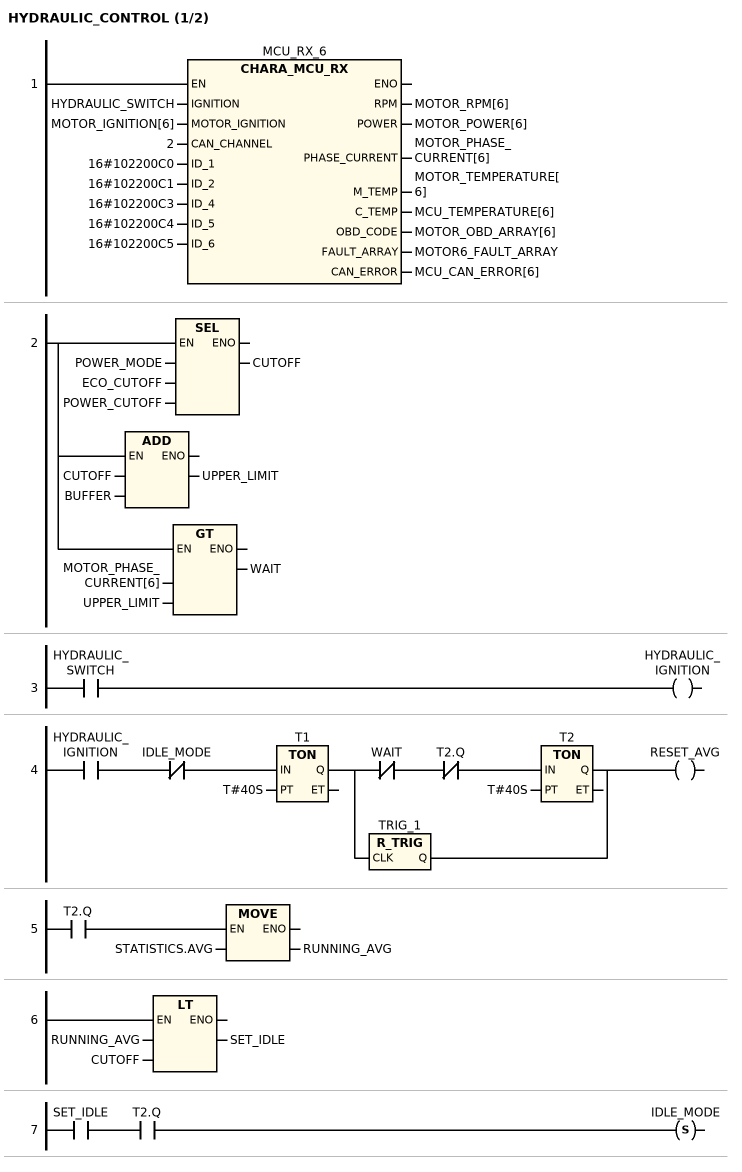
[picture p24: HYDRAULIC_CONTROL (LD)]
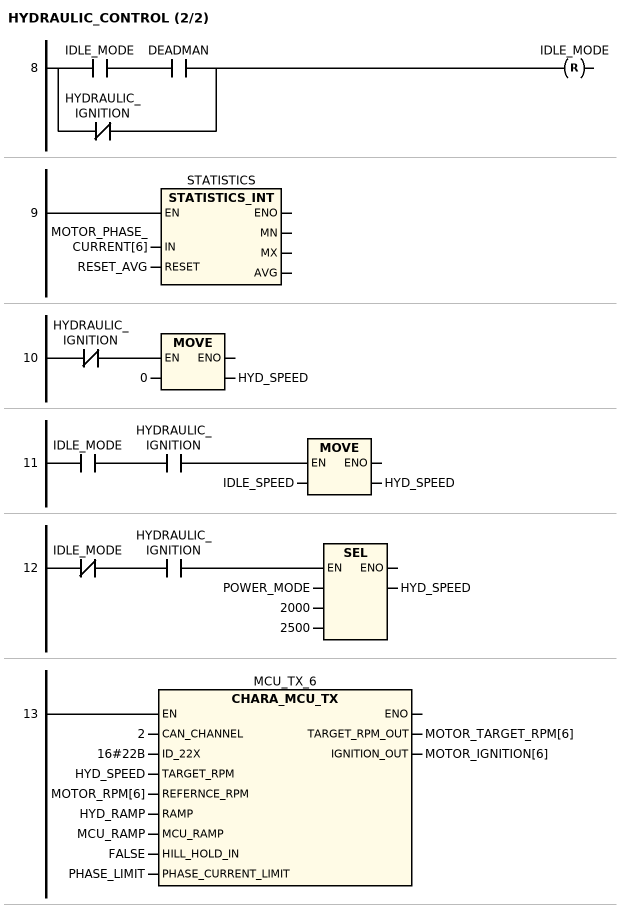
_LD_ (* Ladder Diagram *)
NETWORK 1
	*
		EN --- MCU_RX_6:CHARA_MCU_RX(IGNITION: HYDRAULIC_SWITCH, MOTOR_IGNITION: MOTOR_IGNITION[6], CAN_CHANNEL: 2, ID_1: 16#102200C0, ID_2: 16#102200C1, ID_4: 16#102200C3, ID_5: 16#102200C4, ID_6: 16#102200C5, POWER => MOTOR_POWER[6], PHASE_CURRENT => MOTOR_PHASE_CURRENT[6], M_TEMP => MOTOR_TEMPERATURE[6], C_TEMP => MCU_TEMPERATURE[6], OBD_CODE => MOTOR_OBD_ARRAY[6], FAULT_ARRAY => MOTOR6_FAULT_ARRAY, CAN_ERROR => MCU_CAN_ERROR[6]) => MOTOR_RPM[6]
NETWORK 2
	*
		EN --- SEL(POWER_MODE, ECO_CUTOFF, POWER_CUTOFF) => CUTOFF
		EN --- ADD(CUTOFF, BUFFER) => UPPER_LIMIT
		EN --- GT(MOTOR_PHASE_CURRENT[6], UPPER_LIMIT) => WAIT
NETWORK 3
	[HYDRAULIC_SWITCH] --- (HYDRAULIC_IGNITION)
NETWORK 4
	[HYDRAULIC_IGNITION] - [/IDLE_MODE] - T1:TON(IN: *, PT: T#40S) - { [/WAIT] - [/T2.Q] - T2:TON(IN: *, PT: T#40S) | TRIG_1:R_TRIG(CLK: *) } --- (RESET_AVG)
NETWORK 5
	[T2.Q]
		EN --- MOVE(STATISTICS.AVG) => RUNNING_AVG
NETWORK 6
	*
		EN --- LT(RUNNING_AVG, CUTOFF) => SET_IDLE
NETWORK 7
	[SET_IDLE] - [T2.Q] --- (S IDLE_MODE)
NETWORK 8
	{ [IDLE_MODE] - [DEADMAN] | [/HYDRAULIC_IGNITION] } --- (R IDLE_MODE)
NETWORK 9
	*
		EN --- STATISTICS:STATISTICS_INT(IN: MOTOR_PHASE_CURRENT[6], RESET: RESET_AVG)
NETWORK 10
	[/HYDRAULIC_IGNITION]
		EN --- MOVE(0) => HYD_SPEED
NETWORK 11
	[IDLE_MODE] - [HYDRAULIC_IGNITION]
		EN --- MOVE(IDLE_SPEED) => HYD_SPEED
NETWORK 12
	[/IDLE_MODE] - [HYDRAULIC_IGNITION]
		EN --- SEL(POWER_MODE, 2000, 2500) => HYD_SPEED
NETWORK 13
	*
		EN --- MCU_TX_6:CHARA_MCU_TX(CAN_CHANNEL: 2, ID_22X: 16#22B, TARGET_RPM: HYD_SPEED, REFERNCE_RPM: MOTOR_RPM[6], RAMP: HYD_RAMP, MCU_RAMP: MCU_RAMP, HILL_HOLD_IN: FALSE, PHASE_CURRENT_LIMIT: PHASE_LIMIT, IGNITION_OUT => MOTOR_IGNITION[6]) => MOTOR_TARGET_RPM[6]
_END_LD_
(* the same logic as Structured Text *)
(* Network 1 *)
MCU_RX_6(IGNITION := HYDRAULIC_SWITCH, MOTOR_IGNITION := MOTOR_IGNITION[6], CAN_CHANNEL := 2, ID_1 := 16#102200C0, ID_2 := 16#102200C1, ID_4 := 16#102200C3, ID_5 := 16#102200C4, ID_6 := 16#102200C5);
MOTOR_POWER[6] := MCU_RX_6.POWER;
MOTOR_PHASE_CURRENT[6] := MCU_RX_6.PHASE_CURRENT;
MOTOR_TEMPERATURE[6] := MCU_RX_6.M_TEMP;
MCU_TEMPERATURE[6] := MCU_RX_6.C_TEMP;
MOTOR_OBD_ARRAY[6] := MCU_RX_6.OBD_CODE;
MOTOR6_FAULT_ARRAY := MCU_RX_6.FAULT_ARRAY;
MCU_CAN_ERROR[6] := MCU_RX_6.CAN_ERROR;
MOTOR_RPM[6] := MCU_RX_6.RPM;
(* Network 2 *)
CUTOFF := SEL(POWER_MODE, ECO_CUTOFF, POWER_CUTOFF);
UPPER_LIMIT := CUTOFF + BUFFER;
WAIT := MOTOR_PHASE_CURRENT[6] > UPPER_LIMIT;
(* Network 3 *)
HYDRAULIC_IGNITION := HYDRAULIC_SWITCH;
(* Network 4 *)
T1(IN := HYDRAULIC_IGNITION AND NOT IDLE_MODE, PT := T#40S);
T2(IN := T1.Q AND NOT WAIT AND NOT T2.Q, PT := T#40S);
TRIG_1(CLK := T1.Q);
RESET_AVG := T2.Q OR TRIG_1.Q;
(* Network 5 *)
IF T2.Q THEN
	RUNNING_AVG := STATISTICS.AVG;
END_IF;
(* Network 6 *)
SET_IDLE := RUNNING_AVG < CUTOFF;
(* Network 7 *)
IF SET_IDLE AND T2.Q THEN IDLE_MODE := TRUE; END_IF;
(* Network 8 *)
IF IDLE_MODE AND DEADMAN OR NOT HYDRAULIC_IGNITION THEN IDLE_MODE := FALSE; END_IF;
(* Network 9 *)
STATISTICS(IN := MOTOR_PHASE_CURRENT[6], RESET := RESET_AVG);
(* Network 10 *)
IF NOT HYDRAULIC_IGNITION THEN
	HYD_SPEED := 0;
END_IF;
(* Network 11 *)
IF IDLE_MODE AND HYDRAULIC_IGNITION THEN
	HYD_SPEED := IDLE_SPEED;
END_IF;
(* Network 12 *)
IF NOT IDLE_MODE AND HYDRAULIC_IGNITION THEN
	HYD_SPEED := SEL(POWER_MODE, 2000, 2500);
END_IF;
(* Network 13 *)
MCU_TX_6(CAN_CHANNEL := 2, ID_22X := 16#22B, TARGET_RPM := HYD_SPEED, REFERNCE_RPM := MOTOR_RPM[6], RAMP := HYD_RAMP, MCU_RAMP := MCU_RAMP, HILL_HOLD_IN := FALSE, PHASE_CURRENT_LIMIT := PHASE_LIMIT);
MOTOR_IGNITION[6] := MCU_TX_6.IGNITION_OUT;
MOTOR_TARGET_RPM[6] := MCU_TX_6.TARGET_RPM_OUT;
END_FUNCTION_BLOCK

(* POU MCU/CHARA_MCU_RX, LD *)
FUNCTION_BLOCK CHARA_MCU_RX
(*
Created by: Bhagyesh Unadkat
Date: 11-09-24
Version: 5
Updated by: Karthik
Update date: 08-03-25
Description: This block receives CAN data from CHARA MCU.

		***Updates***
V2
	DC current and POWER added.
V3   
	Added OBD Code and adjusted the fault array accordingly.
	CAN error added to OBD code MSB bit as it is 12-bit value.
V4 
	Taken Motor Ignition as VAR_INPUT to reset RPM AND POWER TO 0
V5
	Converted CURRENT raw values from word to int, and then dividing by 1000.
V6
	Unmerged CAN error and OBD code.
V7
	Making OBD code zero when theres is a CAN error. 

FAULT ARRAY [DATATYPE: BYTE]
[1] MSG-2 BYTE2 and MSG-5 BYTE3		
		BYTE [BIT 0..7]: MSG2BYTE2 (BIT_0 TO BIT_2)------- AND-------- MSG5BYTE3 (BIT_0 TO BIT_4)
[2] MSG 2 :BYTE 7
[3] MSG 5: BYTE 2
[4] MSG 5: BYTE 4
*)
VAR_INPUT
	IGNITION: BOOL;
	MOTOR_IGNITION: BOOL;
	CAN_CHANNEL: BYTE;
	ID_1: DWORD;
	ID_2: DWORD;
	ID_4: DWORD;
	ID_5: DWORD;
	ID_6: DWORD;
END_VAR
VAR_OUTPUT
	RPM: INT;
	POWER: INT;
	PHASE_CURRENT: WORD;
	M_TEMP: BYTE;
	C_TEMP: BYTE;
	OBD_CODE: WORD;
	FAULT_ARRAY: ARRAY [1..4] OF BYTE;
	CAN_ERROR: BOOL;
END_VAR
VAR
	RX_1: RX_CAN;
	RX_2: RX_CAN;
	RX_4: RX_CAN;
	RX_5: RX_CAN;
	RX_6: RX_CAN;
	TIMER_ERROR: TON;

	RPM_WORD: WORD;
	PHASE_WORD: WORD;
	REVERSE_DIRECTION: BOOL;
	DIR_FACTOR: INT;
	DELAY: TON;
	RPM_INT: INT;
	CURRENT_WORD: WORD;
	CURRENT_INT: INT;
	VOLTAGE_INT: INT;
	RPM_SIGNED: INT;
	POWER_INT: INT;
END_VAR
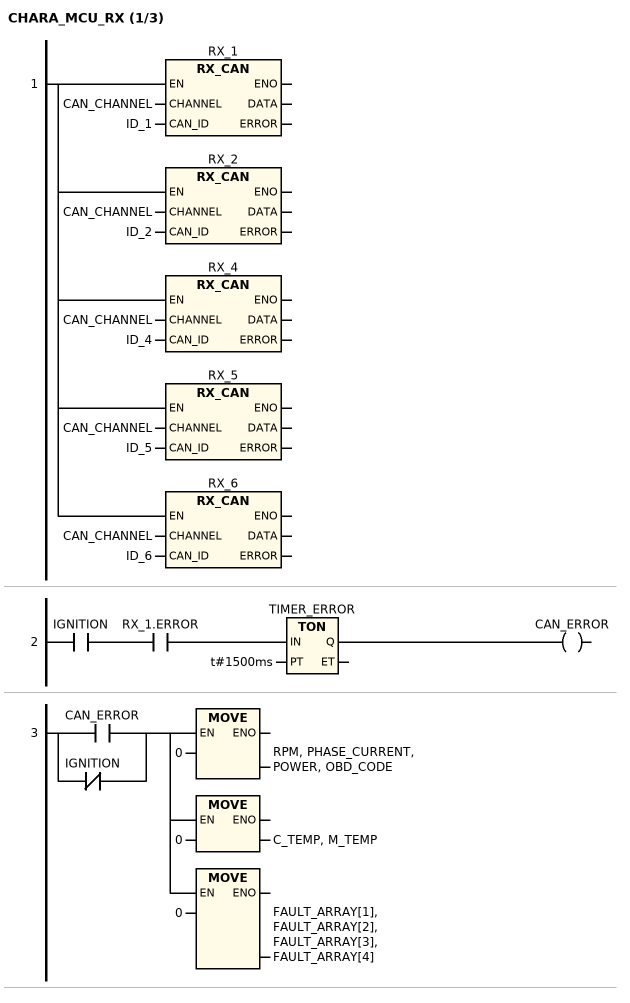
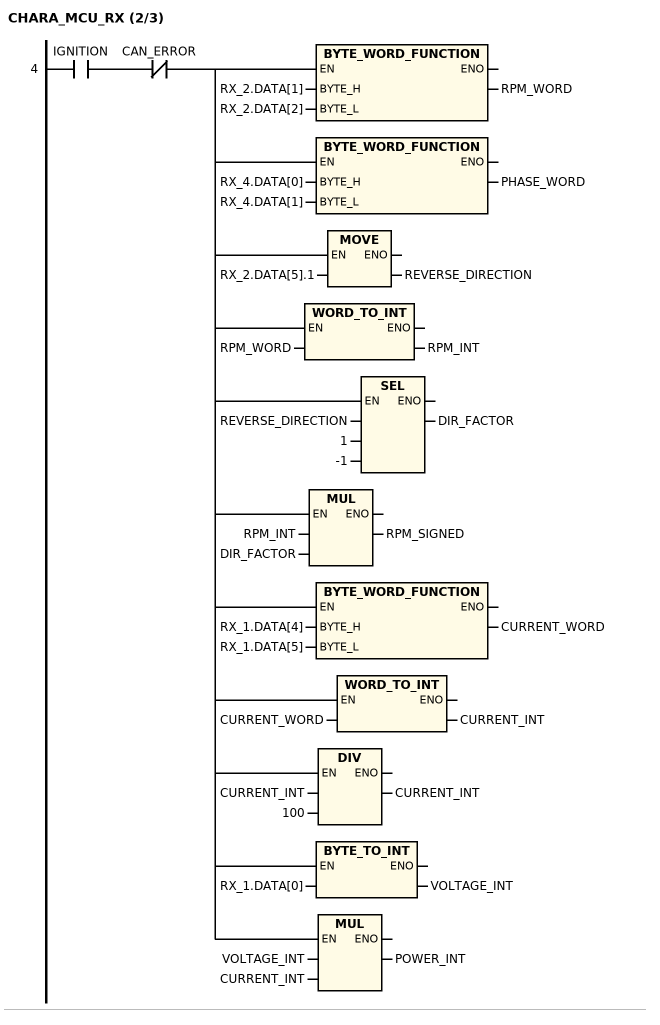
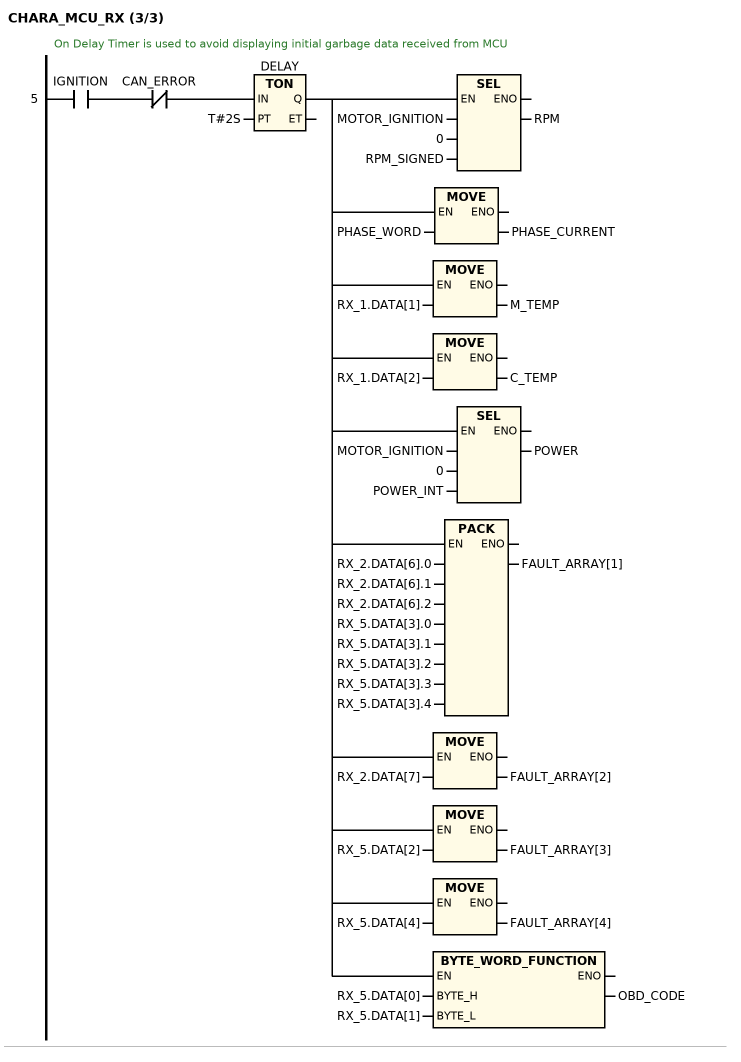
_LD_ (* Ladder Diagram *)
NETWORK 1
	*
		EN --- RX_1:RX_CAN(CHANNEL: CAN_CHANNEL, CAN_ID: ID_1)
		EN --- RX_2:RX_CAN(CHANNEL: CAN_CHANNEL, CAN_ID: ID_2)
		EN --- RX_4:RX_CAN(CHANNEL: CAN_CHANNEL, CAN_ID: ID_4)
		EN --- RX_5:RX_CAN(CHANNEL: CAN_CHANNEL, CAN_ID: ID_5)
		EN --- RX_6:RX_CAN(CHANNEL: CAN_CHANNEL, CAN_ID: ID_6)
NETWORK 2
	[IGNITION] - [RX_1.ERROR] - TIMER_ERROR:TON(IN: *, PT: t#1500ms) --- (CAN_ERROR)
NETWORK 3
	{ [CAN_ERROR] | [/IGNITION] }
		EN --- MOVE(0) => RPM, PHASE_CURRENT, POWER, OBD_CODE
		EN --- MOVE(0) => C_TEMP, M_TEMP
		EN --- MOVE(0) => FAULT_ARRAY[1], FAULT_ARRAY[2], FAULT_ARRAY[3], FAULT_ARRAY[4]
NETWORK 4
	[IGNITION] - [/CAN_ERROR]
		EN --- BYTE_WORD_FUNCTION(BYTE_H: RX_2.DATA[1], BYTE_L: RX_2.DATA[2]) => RPM_WORD
		EN --- BYTE_WORD_FUNCTION(BYTE_H: RX_4.DATA[0], BYTE_L: RX_4.DATA[1]) => PHASE_WORD
		EN --- MOVE(RX_2.DATA[5].1) => REVERSE_DIRECTION
		EN --- WORD_TO_INT(RPM_WORD) => RPM_INT
		EN --- SEL(REVERSE_DIRECTION, 1, -1) => DIR_FACTOR
		EN --- MUL(RPM_INT, DIR_FACTOR) => RPM_SIGNED
		EN --- BYTE_WORD_FUNCTION(BYTE_H: RX_1.DATA[4], BYTE_L: RX_1.DATA[5]) => CURRENT_WORD
		EN --- WORD_TO_INT(CURRENT_WORD) => CURRENT_INT
		EN --- DIV(CURRENT_INT, 100) => CURRENT_INT
		EN --- BYTE_TO_INT(RX_1.DATA[0]) => VOLTAGE_INT
		EN --- MUL(VOLTAGE_INT, CURRENT_INT) => POWER_INT
NETWORK 5 (* On Delay Timer is used to avoid displaying initial garbage data received from MCU *)
	[IGNITION] - [/CAN_ERROR] - DELAY:TON(IN: *, PT: T#2S)
		EN --- SEL(MOTOR_IGNITION, 0, RPM_SIGNED) => RPM
		EN --- MOVE(PHASE_WORD) => PHASE_CURRENT
		EN --- MOVE(RX_1.DATA[1]) => M_TEMP
		EN --- MOVE(RX_1.DATA[2]) => C_TEMP
		EN --- SEL(MOTOR_IGNITION, 0, POWER_INT) => POWER
		EN --- PACK(RX_2.DATA[6].0, RX_2.DATA[6].1, RX_2.DATA[6].2, RX_5.DATA[3].0, RX_5.DATA[3].1, RX_5.DATA[3].2, RX_5.DATA[3].3, RX_5.DATA[3].4) => FAULT_ARRAY[1]
		EN --- MOVE(RX_2.DATA[7]) => FAULT_ARRAY[2]
		EN --- MOVE(RX_5.DATA[2]) => FAULT_ARRAY[3]
		EN --- MOVE(RX_5.DATA[4]) => FAULT_ARRAY[4]
		EN --- BYTE_WORD_FUNCTION(BYTE_H: RX_5.DATA[0], BYTE_L: RX_5.DATA[1]) => OBD_CODE
_END_LD_
(* the same logic as Structured Text *)
(* Network 1 *)
RX_1(CHANNEL := CAN_CHANNEL, CAN_ID := ID_1);
RX_2(CHANNEL := CAN_CHANNEL, CAN_ID := ID_2);
RX_4(CHANNEL := CAN_CHANNEL, CAN_ID := ID_4);
RX_5(CHANNEL := CAN_CHANNEL, CAN_ID := ID_5);
RX_6(CHANNEL := CAN_CHANNEL, CAN_ID := ID_6);
(* Network 2 *)
TIMER_ERROR(IN := IGNITION AND RX_1.ERROR, PT := t#1500ms);
CAN_ERROR := TIMER_ERROR.Q;
(* Network 3: see the listing above *)
(* Network 4 *)
IF IGNITION AND NOT CAN_ERROR THEN
	RPM_WORD := BYTE_WORD_FUNCTION(BYTE_H := RX_2.DATA[1], BYTE_L := RX_2.DATA[2]);
	PHASE_WORD := BYTE_WORD_FUNCTION(BYTE_H := RX_4.DATA[0], BYTE_L := RX_4.DATA[1]);
	REVERSE_DIRECTION := RX_2.DATA[5].1;
	RPM_INT := WORD_TO_INT(RPM_WORD);
	DIR_FACTOR := SEL(REVERSE_DIRECTION, 1, -1);
	RPM_SIGNED := RPM_INT * DIR_FACTOR;
	CURRENT_WORD := BYTE_WORD_FUNCTION(BYTE_H := RX_1.DATA[4], BYTE_L := RX_1.DATA[5]);
	CURRENT_INT := WORD_TO_INT(CURRENT_WORD);
	CURRENT_INT := CURRENT_INT / 100;
	VOLTAGE_INT := BYTE_TO_INT(RX_1.DATA[0]);
	POWER_INT := VOLTAGE_INT * CURRENT_INT;
END_IF;
(* Network 5 *)
DELAY(IN := IGNITION AND NOT CAN_ERROR, PT := T#2S);
IF DELAY.Q THEN
	RPM := SEL(MOTOR_IGNITION, 0, RPM_SIGNED);
	PHASE_CURRENT := PHASE_WORD;
	M_TEMP := RX_1.DATA[1];
	C_TEMP := RX_1.DATA[2];
	POWER := SEL(MOTOR_IGNITION, 0, POWER_INT);
	FAULT_ARRAY[1] := PACK(RX_2.DATA[6].0, RX_2.DATA[6].1, RX_2.DATA[6].2, RX_5.DATA[3].0, RX_5.DATA[3].1, RX_5.DATA[3].2, RX_5.DATA[3].3, RX_5.DATA[3].4);
	FAULT_ARRAY[2] := RX_2.DATA[7];
	FAULT_ARRAY[3] := RX_5.DATA[2];
	FAULT_ARRAY[4] := RX_5.DATA[4];
	OBD_CODE := BYTE_WORD_FUNCTION(BYTE_H := RX_5.DATA[0], BYTE_L := RX_5.DATA[1]);
END_IF;
END_FUNCTION_BLOCK

(* POU MCU/CHARA_MCU_TX, LD *)
FUNCTION_BLOCK CHARA_MCU_TX
(*
Created by: Bhagyesh Unadkat
Date: Sep 11, 2024
Version: 4
Updated by: Bhagyesh
Update date: Dec 13, 2024
Description: This block transmits CAN data to the CHARA MCU to control the motor.

NOTE:  BIG ENDIAN FORMAT

Byte0 & Byte1: Signed RPM Big Endian format (-6000 to 6000)
Byte2: Ignition State =  0 & 1 (OFF and ON respectively)
Byte3: Phase Current Limit (%) = 0 - 100
Byte4: Regen (%) = 0 - 100 (Not configured yet)
Byte5: Acceleration time (s) = 1 unit is 100ms
Byte6: Deceleration time (s) =  1 unit is 100ms

CAN ID X value for the different Node ID:
41 - 9		42 - A 		43-B
	
	***UPDATES***
V2:
1. RPM transmit delay has been added after Ignition turns on..
2. CAN_TX block has been changerd to CAN_TX_ENH.
3. Temporary Phase current limit has been added to var input
V3
1. Added Ignition state bit as VAR_OUTPUT.
V4
1. UPDATED AVG RPM TO 75 TO HOLD ON THE MCU.
2. RPM DELAY TIME REDUCED TO 250MS
*)
VAR_INPUT
	CAN_CHANNEL: BYTE;
	ID_22X: DWORD;
	TARGET_RPM: INT;
	REFERNCE_RPM: INT;
	RAMP: INT;
	MCU_RAMP: BYTE;
	HILL_HOLD_IN: BOOL;
	PHASE_CURRENT_LIMIT: BYTE;
END_VAR
VAR
	IGNITION_ON: BOOL;
	IGNITION_STATE: BYTE;
	HOLD_ON: BOOL;
	ABS_RPM: INT;
	RPM_RAMP: RAMP_INT;
	WB_TARGET_RPM: WORD_BYTE_CONVERSION;
	PACK_TX: PACK_BYTES;
	TX: CAN_TX_ENH;
	RPM_DELAY: TON;
	TIMER: TON;
END_VAR
VAR_OUTPUT
	TARGET_RPM_OUT: INT;
	IGNITION_OUT: BOOL;
END_VAR
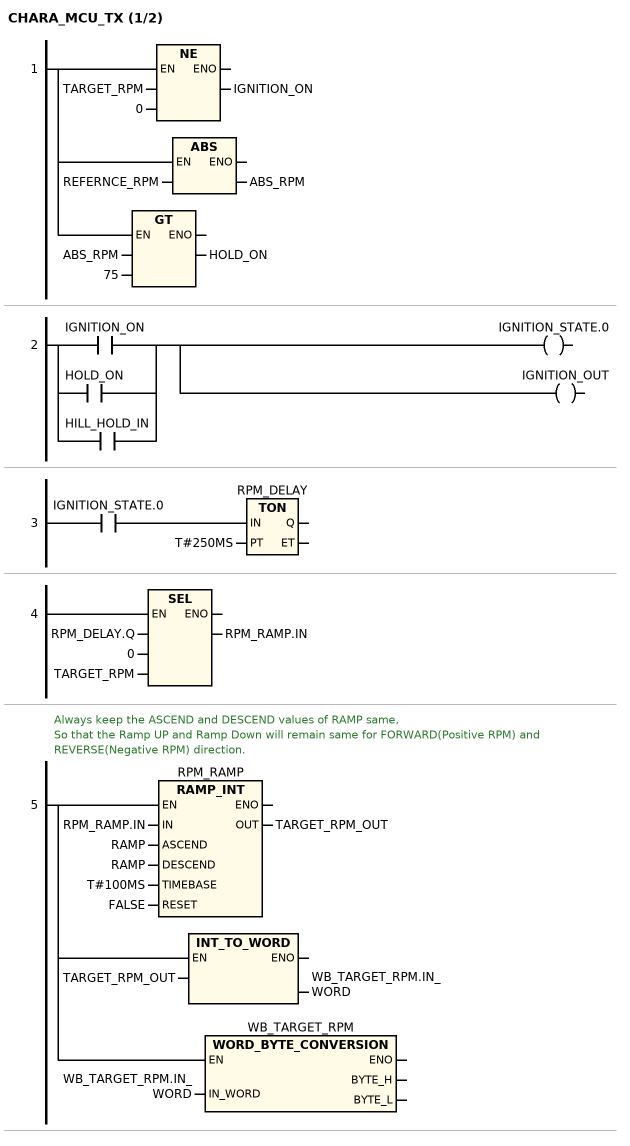
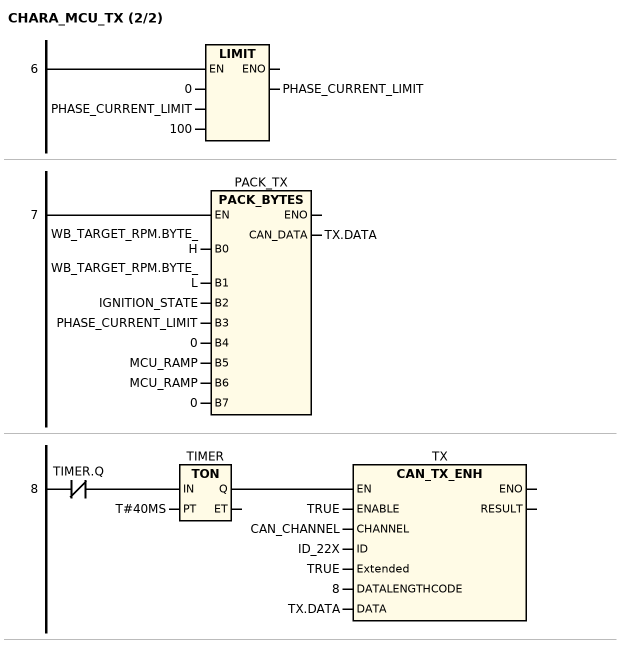
_LD_ (* Ladder Diagram *)
NETWORK 1
	*
		EN --- NE(TARGET_RPM, 0) => IGNITION_ON
		EN --- ABS(REFERNCE_RPM) => ABS_RPM
		EN --- GT(ABS_RPM, 75) => HOLD_ON
NETWORK 2
	{ [IGNITION_ON] | [HOLD_ON] | [HILL_HOLD_IN] } --- (IGNITION_STATE.0) (IGNITION_OUT)
NETWORK 3
	[IGNITION_STATE.0] - RPM_DELAY:TON(IN: *, PT: T#250MS)
NETWORK 4
	*
		EN --- SEL(RPM_DELAY.Q, 0, TARGET_RPM) => RPM_RAMP.IN
NETWORK 5 (* Always keep the ASCEND and DESCEND values of RAMP same, / So that the Ramp UP and Ramp Down will remain same for FORWARD(Positive RPM) and REVERSE(Negative RPM) direction. *)
	*
		EN --- RPM_RAMP:RAMP_INT(IN: RPM_RAMP.IN, ASCEND: RAMP, DESCEND: RAMP, TIMEBASE: T#100MS, RESET: FALSE) => TARGET_RPM_OUT
		EN --- INT_TO_WORD(TARGET_RPM_OUT) => WB_TARGET_RPM.IN_WORD
		EN --- WB_TARGET_RPM:WORD_BYTE_CONVERSION(IN_WORD: WB_TARGET_RPM.IN_WORD)
NETWORK 6
	*
		EN --- LIMIT(0, PHASE_CURRENT_LIMIT, 100) => PHASE_CURRENT_LIMIT
NETWORK 7
	*
		EN --- PACK_TX:PACK_BYTES(B0: WB_TARGET_RPM.BYTE_H, B1: WB_TARGET_RPM.BYTE_L, B2: IGNITION_STATE, B3: PHASE_CURRENT_LIMIT, B4: 0, B5: MCU_RAMP, B6: MCU_RAMP, B7: 0) => TX.DATA
NETWORK 8
	[/TIMER.Q] - TIMER:TON(IN: *, PT: T#40MS)
		EN --- TX:CAN_TX_ENH(ENABLE: TRUE, CHANNEL: CAN_CHANNEL, ID: ID_22X, Extended: TRUE, DATALENGTHCODE: 8, DATA: TX.DATA)
_END_LD_
(* the same logic as Structured Text *)
(* Network 1 *)
IGNITION_ON := TARGET_RPM <> 0;
ABS_RPM := ABS(REFERNCE_RPM);
HOLD_ON := ABS_RPM > 75;
(* Network 2 *)
IGNITION_STATE.0 := IGNITION_ON OR HOLD_ON OR HILL_HOLD_IN;
IGNITION_OUT := IGNITION_STATE.0;
(* Network 3 *)
RPM_DELAY(IN := IGNITION_STATE.0, PT := T#250MS);
(* Network 4 *)
RPM_RAMP.IN := SEL(RPM_DELAY.Q, 0, TARGET_RPM);
(* Network 5: Always keep the ASCEND and DESCEND values of RAMP same, / So that the Ramp UP and Ramp Down will remain same for FORWARD(Positive RPM) and REVERSE(Negative RPM) direction. *)
RPM_RAMP(IN := RPM_RAMP.IN, ASCEND := RAMP, DESCEND := RAMP, TIMEBASE := T#100MS, RESET := FALSE);
TARGET_RPM_OUT := RPM_RAMP.OUT;
WB_TARGET_RPM.IN_WORD := INT_TO_WORD(TARGET_RPM_OUT);
WB_TARGET_RPM(IN_WORD := WB_TARGET_RPM.IN_WORD);
(* Network 6 *)
PHASE_CURRENT_LIMIT := LIMIT(0, PHASE_CURRENT_LIMIT, 100);
(* Network 7 *)
PACK_TX(B0 := WB_TARGET_RPM.BYTE_H, B1 := WB_TARGET_RPM.BYTE_L, B2 := IGNITION_STATE, B3 := PHASE_CURRENT_LIMIT, B4 := 0, B5 := MCU_RAMP, B6 := MCU_RAMP, B7 := 0);
TX.DATA := PACK_TX.CAN_DATA;
(* Network 8 *)
TIMER(IN := NOT TIMER.Q, PT := T#40MS);
IF TIMER.Q THEN
	TX(ENABLE := TRUE, CHANNEL := CAN_CHANNEL, ID := ID_22X, Extended := TRUE, DATALENGTHCODE := 8, DATA := TX.DATA);
END_IF;
END_FUNCTION_BLOCK

(* POU FB_LIBRARY/WORD_BYTE_CONVERSION, FBD *)
FUNCTION_BLOCK WORD_BYTE_CONVERSION
(*
Created by: Bhagyesh Unadkat
Date: 29-03-24
Version: 1
Updated by:
Update date:
Description: This block converts the WORD data into two BYTEs
*)
VAR_INPUT
	IN_WORD: WORD;
END_VAR
VAR_OUTPUT
	BYTE_H: BYTE;
	BYTE_L: BYTE;
END_VAR
VAR
END_VAR
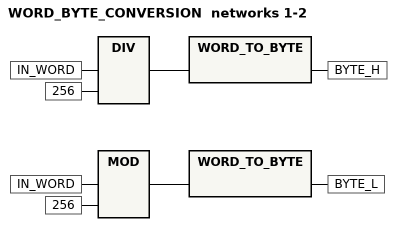
_FBD_ (* Function Block Diagram *)
NETWORK 1
	WORD_TO_BYTE(DIV(IN_WORD, 256)) => BYTE_H
NETWORK 2
	WORD_TO_BYTE(MOD(IN_WORD, 256)) => BYTE_L
_END_FBD_
(* the same logic as Structured Text *)
(* Network 1 *)
BYTE_H := WORD_TO_BYTE(IN_WORD / 256);
(* Network 2 *)
BYTE_L := WORD_TO_BYTE(IN_WORD MOD 256);
END_FUNCTION_BLOCK

(* POU FB_LIBRARY/PACK_BYTES, ST *)
FUNCTION_BLOCK PACK_BYTES
(*
Created by: Bhagyesh Unadkat
Date: 29-03-24
Version: 1
Updated by:
Update date:
Description: This block merges 8 bytes of data into 1 CAN data array.
*)
VAR_INPUT
	B0: BYTE;
	B1: BYTE;
	B2: BYTE;
	B3: BYTE;
	B4: BYTE;
	B5: BYTE;
	B6: BYTE;
	B7: BYTE;
END_VAR
VAR_OUTPUT
	CAN_DATA: ARRAY [0..7] OF BYTE;
END_VAR
CAN_DATA[0]:= B0;
CAN_DATA[1]:= B1;
CAN_DATA[2]:= B2;
CAN_DATA[3]:= B3;
CAN_DATA[4]:= B4;
CAN_DATA[5]:= B5;
CAN_DATA[6]:= B6;
CAN_DATA[7]:= B7;
END_FUNCTION_BLOCK

(* POU PROGRAM_FBs/ARM_LOGIC, LD *)
FUNCTION_BLOCK ARM_LOGIC
VAR_INPUT
	ARM_INPUT: BOOL;
	DISARM: BOOL;
	POST_IN: BOOL;
END_VAR
VAR_OUTPUT
	ARM: BOOL;
	ARMLED: BOOL;
END_VAR
VAR
	DELAY: TON;
	S1: BOOL;
	S2: BOOL;
	BLINKY: BLINK;
END_VAR
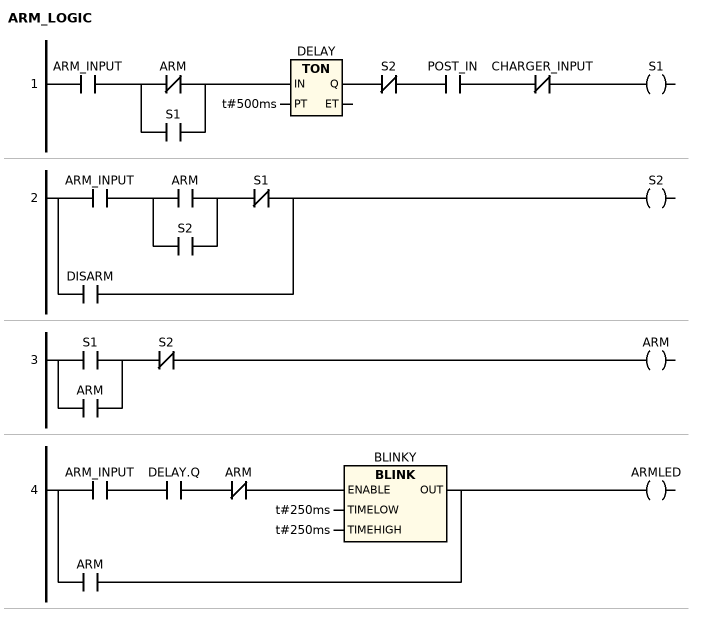
_LD_ (* Ladder Diagram *)
NETWORK 1
	[ARM_INPUT] - { [/ARM] | [S1] } - DELAY:TON(IN: *, PT: t#500ms) - [/S2] - [POST_IN] - [/CHARGER_INPUT] --- (S1)
NETWORK 2
	{ [ARM_INPUT] - { [ARM] | [S2] } - [/S1] | [DISARM] } --- (S2)
NETWORK 3
	{ [S1] | [ARM] } - [/S2] --- (ARM)
NETWORK 4
	{ [ARM_INPUT] - [DELAY.Q] - [/ARM] - BLINKY:BLINK(ENABLE: *, TIMELOW: t#250ms, TIMEHIGH: t#250ms) | [ARM] } --- (ARMLED)
_END_LD_
(* the same logic as Structured Text *)
(* Network 1 *)
DELAY(IN := ARM_INPUT AND (NOT ARM OR S1), PT := t#500ms);
S1 := DELAY.Q AND NOT S2 AND POST_IN AND NOT CHARGER_INPUT;
(* Network 2 *)
S2 := ARM_INPUT AND (ARM OR S2) AND NOT S1 OR DISARM;
(* Network 3 *)
ARM := (S1 OR ARM) AND NOT S2;
(* Network 4 *)
BLINKY(ENABLE := ARM_INPUT AND DELAY.Q AND NOT ARM, TIMELOW := t#250ms, TIMEHIGH := t#250ms);
ARMLED := BLINKY.OUT OR ARM;
END_FUNCTION_BLOCK

(* POU PROGRAM_FBs/DRIVE_LOGIC, LD *)
FUNCTION_BLOCK DRIVE_LOGIC
VAR_INPUT
	JX: INT;
	JY: INT;
	LEFT_BUTTON: BOOL;
	JOY_ORIGIN: BOOL;
	EM_SWITCH_IN: BOOL;
	OVER_TEMP: BOOL;
END_VAR
VAR_OUTPUT
	JX_1: INT;
	JY_1: INT;
	DISARM: BOOL;
	EM_BRAKE_OUT: BOOL;
	DRIVE_ERROR: BOOL;
END_VAR
VAR
	SLEEP_TIMER: TON;
	ON_DELAY: TON;
	APPLY_EM: BOOL;
	LOW_RPM: BOOL;
	EMFB_ERROR: BOOL;
END_VAR
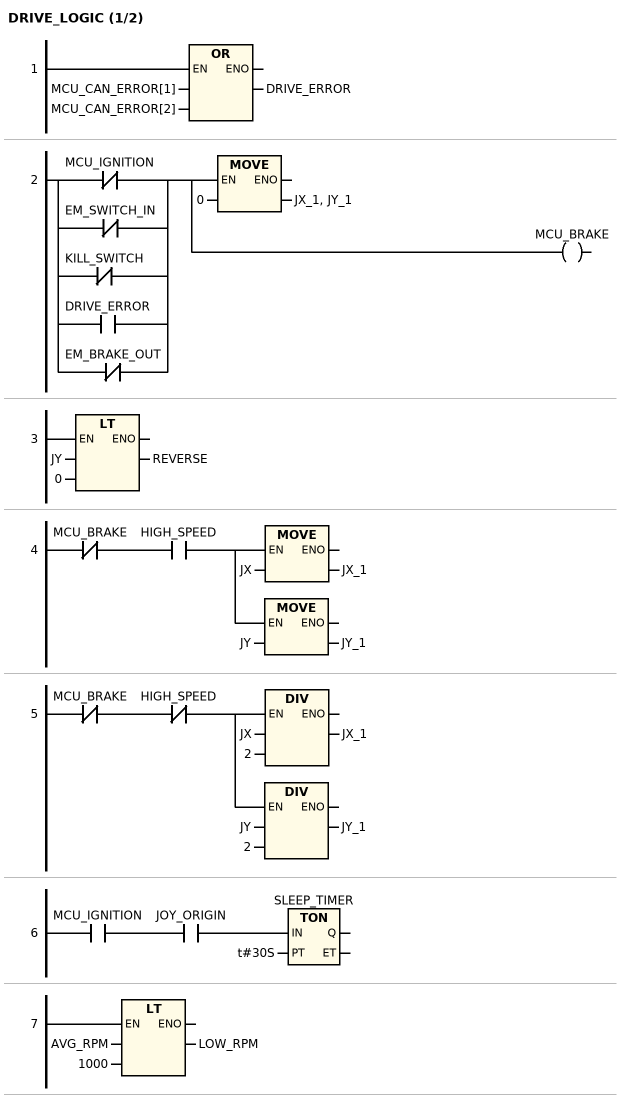
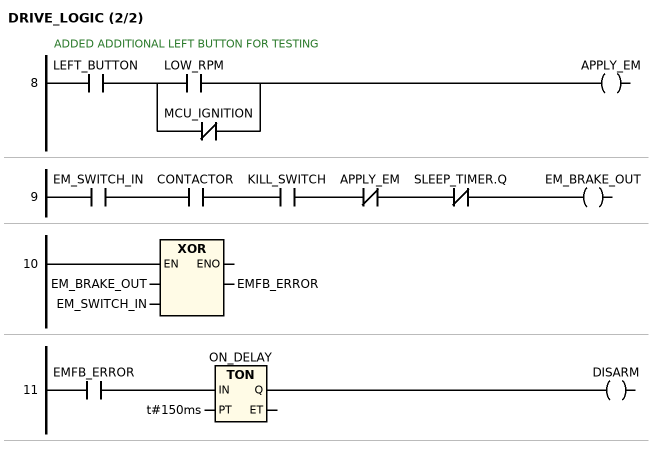
_LD_ (* Ladder Diagram *)
NETWORK 1
	*
		EN --- OR(MCU_CAN_ERROR[1], MCU_CAN_ERROR[2]) => DRIVE_ERROR
NETWORK 2
	{ [/MCU_IGNITION] | [/EM_SWITCH_IN] | [/KILL_SWITCH] | [DRIVE_ERROR] | [/EM_BRAKE_OUT] } --- (MCU_BRAKE)
		EN --- MOVE(0) => JX_1, JY_1
NETWORK 3
	*
		EN --- LT(JY, 0) => REVERSE
NETWORK 4
	[/MCU_BRAKE] - [HIGH_SPEED]
		EN --- MOVE(JX) => JX_1
		EN --- MOVE(JY) => JY_1
NETWORK 5
	[/MCU_BRAKE] - [/HIGH_SPEED]
		EN --- DIV(JX, 2) => JX_1
		EN --- DIV(JY, 2) => JY_1
NETWORK 6
	[MCU_IGNITION] - [JOY_ORIGIN] - SLEEP_TIMER:TON(IN: *, PT: t#30S)
NETWORK 7
	*
		EN --- LT(AVG_RPM, 1000) => LOW_RPM
NETWORK 8 (* ADDED ADDITIONAL LEFT BUTTON FOR TESTING *)
	[LEFT_BUTTON] - { [LOW_RPM] | [/MCU_IGNITION] } --- (APPLY_EM)
NETWORK 9
	[EM_SWITCH_IN] - [CONTACTOR] - [KILL_SWITCH] - [/APPLY_EM] - [/SLEEP_TIMER.Q] --- (EM_BRAKE_OUT)
NETWORK 10
	*
		EN --- XOR(EM_BRAKE_OUT, EM_SWITCH_IN) => EMFB_ERROR
NETWORK 11
	[EMFB_ERROR] - ON_DELAY:TON(IN: *, PT: t#150ms) --- (DISARM)
_END_LD_
(* the same logic as Structured Text *)
(* Network 1 *)
DRIVE_ERROR := MCU_CAN_ERROR[1] OR MCU_CAN_ERROR[2];
(* Network 2: see the listing above *)
(* Network 3 *)
REVERSE := JY < 0;
(* Network 4 *)
IF NOT MCU_BRAKE AND HIGH_SPEED THEN
	JX_1 := JX;
	JY_1 := JY;
END_IF;
(* Network 5 *)
IF NOT MCU_BRAKE AND NOT HIGH_SPEED THEN
	JX_1 := JX / 2;
	JY_1 := JY / 2;
END_IF;
(* Network 6 *)
SLEEP_TIMER(IN := MCU_IGNITION AND JOY_ORIGIN, PT := t#30S);
(* Network 7 *)
LOW_RPM := AVG_RPM < 1000;
(* Network 8 *)
APPLY_EM := LEFT_BUTTON AND (LOW_RPM OR NOT MCU_IGNITION);
(* Network 9 *)
EM_BRAKE_OUT := EM_SWITCH_IN AND CONTACTOR AND KILL_SWITCH AND NOT APPLY_EM AND NOT SLEEP_TIMER.Q;
(* Network 10 *)
EMFB_ERROR := EM_BRAKE_OUT XOR EM_SWITCH_IN;
(* Network 11 *)
ON_DELAY(IN := EMFB_ERROR, PT := t#150ms);
DISARM := ON_DELAY.Q;
END_FUNCTION_BLOCK

(* POU PROGRAM_FBs/THROTTLE_LOGIC, LD *)
FUNCTION_BLOCK THROTTLE_LOGIC
(*
Author: Bhagyesh
Description: This function block takes the joystick input from the RunLogic block and calculates the throttle for each side of the motors based on the turning logic.
This function block also implements the Zero degree turn.
*)
VAR_INPUT
	JX_IN: INT;
	JY_IN: INT;
	MCUBRAKE: BOOL;
	RPM_FACTOR_IN: INT;
END_VAR
VAR_OUTPUT
	THR_L: INT;
	THR_R: INT;
END_VAR
VAR
	THR_1: INT;
	THR_2: INT;
	THR_R_INTER: INT;
	SET_FWD: BOOL;
	SET_REV: BOOL;
	SET_RIGHT_ZERO: BOOL;
	SET_LEFT_ZERO: BOOL;

	JOY_ORIGIN: BOOL;
	FWD: BOOL;
	REV: BOOL;
	RIGHT_ZERO: BOOL;
	LEFT_ZERO: BOOL;
END_VAR
VAR CONSTANT

END_VAR
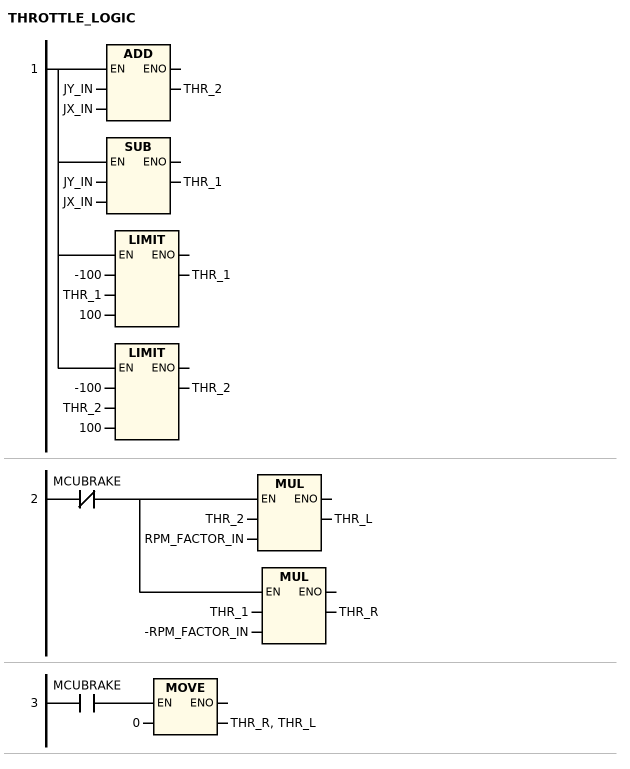
_LD_ (* Ladder Diagram *)
NETWORK 1
	*
		EN --- ADD(JY_IN, JX_IN) => THR_2
		EN --- SUB(JY_IN, JX_IN) => THR_1
		EN --- LIMIT(-100, THR_1, 100) => THR_1
		EN --- LIMIT(-100, THR_2, 100) => THR_2
NETWORK 2
	[/MCUBRAKE]
		EN --- MUL(THR_2, RPM_FACTOR_IN) => THR_L
		EN --- MUL(THR_1, -RPM_FACTOR_IN) => THR_R
NETWORK 3
	[MCUBRAKE]
		EN --- MOVE(0) => THR_R, THR_L
_END_LD_
(* the same logic as Structured Text *)
(* Network 1 *)
THR_2 := JY_IN + JX_IN;
THR_1 := JY_IN - JX_IN;
THR_1 := LIMIT(-100, THR_1, 100);
THR_2 := LIMIT(-100, THR_2, 100);
(* Network 2 *)
IF NOT MCUBRAKE THEN
	THR_L := THR_2 * RPM_FACTOR_IN;
	THR_R := THR_1 * (-RPM_FACTOR_IN);
END_IF;
(* Network 3: see the listing above *)
END_FUNCTION_BLOCK

(* POU TELEMATICS, LD *)
PROGRAM TELEMATICS
VAR
	TX_300: CAN_TX;
	TX_301: CAN_TX;
	TX_303: CAN_TX;
	TX_305: CAN_TX;
	TX_306: CAN_TX;
   	TX_307: CAN_TX;
	TX_308: CAN_TX;
	TX_310: CAN_TX;
	TX_311: CAN_TX;
	TX_312: CAN_TX;
	TX_313: CAN_TX;
	TX_31A: CAN_TX;
	TX_31B: CAN_TX;

	TX_400: CAN_TX;
	TX_401: CAN_TX;
	TX_403: CAN_TX;
	TX_405: CAN_TX;
	TX_406: CAN_TX;
   	TX_407: CAN_TX;
	TX_408: CAN_TX;
	TX_410: CAN_TX;
	TX_411: CAN_TX;
	TX_412: CAN_TX;
	TX_413: CAN_TX;
	TX_41A: CAN_TX;
	TX_41B: CAN_TX;
	TX_262: CAN_TX;

	RX_7F0: RX_CAN;
	RX_450: RX_CAN;

	PACK_301: PACK_BYTES;
	PACK_303: PACK_BYTES;
	PACK_305: PACK_BYTES;
	PACK_306: PACK_BYTES;
	PACK_308: PACK_BYTES;
	PACK_311: PACK_BYTES;
	PACK_313: PACK_BYTES;
	PACK_31B: PACK_BYTES;
	PACK_262: PACK_BYTES;

	WB_BATTERY1_POWER: WORD_BYTE_CONVERSION;
	WB_RPM_1: WORD_BYTE_CONVERSION;
	WB_POWER_1: WORD_BYTE_CONVERSION;
	WB_PHASE_1: WORD_BYTE_CONVERSION;
	WB_TARGET_RPM_1: WORD_BYTE_CONVERSION;

	WB_BATTERY2_POWER: WORD_BYTE_CONVERSION;
	WB_RPM_2: WORD_BYTE_CONVERSION;
	WB_POWER_2: WORD_BYTE_CONVERSION;
	WB_PHASE_2: WORD_BYTE_CONVERSION;
	WB_TARGET_RPM_2: WORD_BYTE_CONVERSION;

	WB_RPM_6: WORD_BYTE_CONVERSION;
	WB_POWER_6: WORD_BYTE_CONVERSION;
	WB_PHASE_6: WORD_BYTE_CONVERSION;
	WB_TARGET_RPM_6: WORD_BYTE_CONVERSION;
	WB_FAULTS_6: WORD_BYTE_CONVERSION;

	WB_RUNTIME: WORD_BYTE_CONVERSION;

	DATA_LOG_ERROR: BOOL;
	DWIN_CAN_ERROR: BOOL;
	TIMER_DATALOG: TON;
	TIMER_DWIN: TON;
	TIMER_TX: TON;

	WD_BATTERY1_FULLCHARGE_MIN: WORD;
	WD_BATTERY2_FULLCHARGE_MIN: WORD;
	WB_FULLCHARGE1_MIN: WORD_BYTE_CONVERSION;
	WB_FULLCHARGE2_MIN: WORD_BYTE_CONVERSION;

	WB_OBD_1: WORD_BYTE_CONVERSION;
	WB_OBD_2: WORD_BYTE_CONVERSION;
	WB_OBD_6: WORD_BYTE_CONVERSION;

	WB_HYDL_UP_TIME: WORD_BYTE_CONVERSION;
	WB_TRIP_KM: WORD_BYTE_CONVERSION;
	WB_ODO_METERS: DWORD_BYTE_CONVERSION;
	WB_RUNTIME_MIN: DWORD_BYTE_CONVERSION;
	TIMER_TX_1: TON;
	TIMER_TX_2: TON;
	RX_3A0: RX_CAN;
	TRIP: WORD_BYTE_CONVERSION;
	OBD1_INT: INT;
	OBD1_BYTE: BYTE;
	OBD2_INT: INT;
	OBD2_BYTE: BYTE;
	OBD6_INT: INT;
	OBD6_BYTE: BYTE;
	WB_HYDL_UPTIME: DWORD_BYTE_CONVERSION;
	WB_VEHICLE_UPTIME: DWORD_BYTE_CONVERSION;
	TX_409: CAN_TX;
	PACK_409: PACK_BYTES;
	WB_VEHICLE_UPTIME_LT: DWORD_BYTE_CONVERSION;
END_VAR
VAR CONSTANT
	META_FRAME: ARRAY [0..7] OF BYTE := 18,1,1,0,0,0,0,0; (*GLX_PR, KEY1, VX,VY,VZ*)
	CAN_CHANNEL: BYTE := 1;
END_VAR
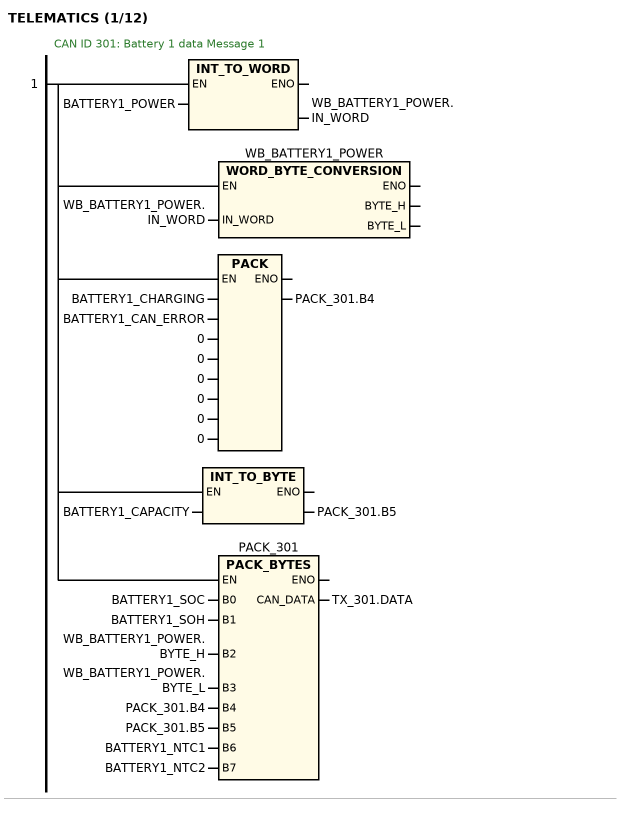
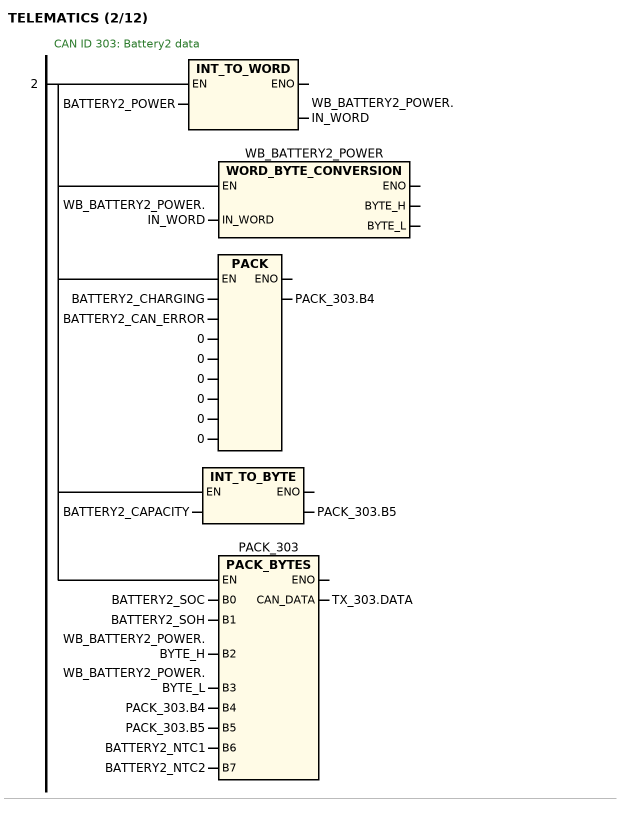
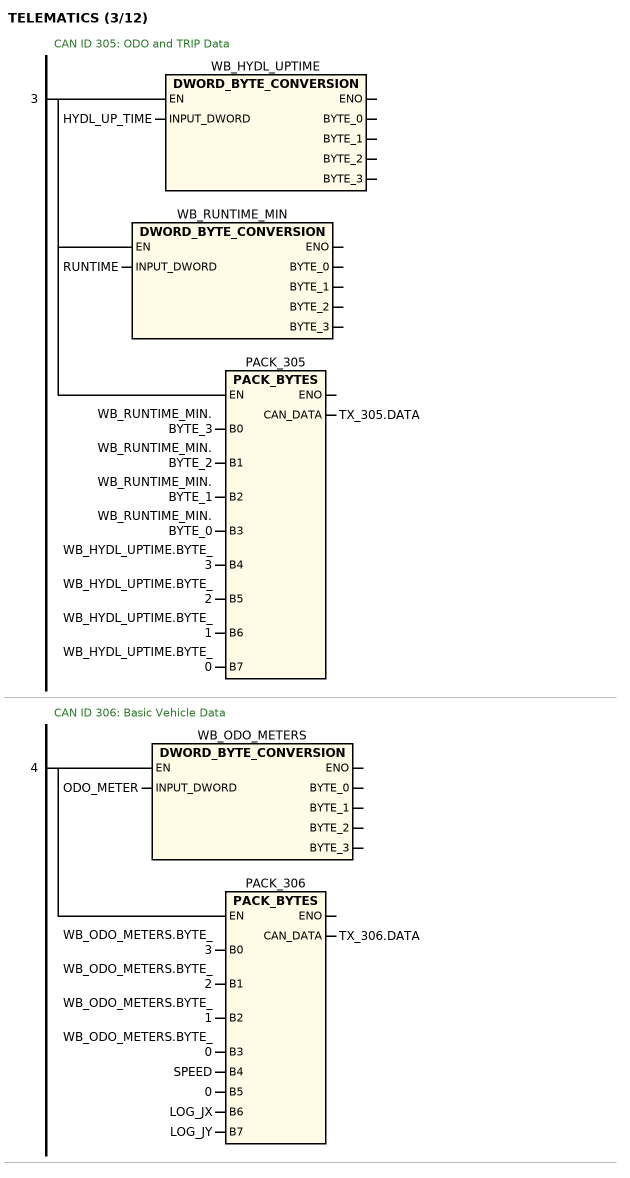
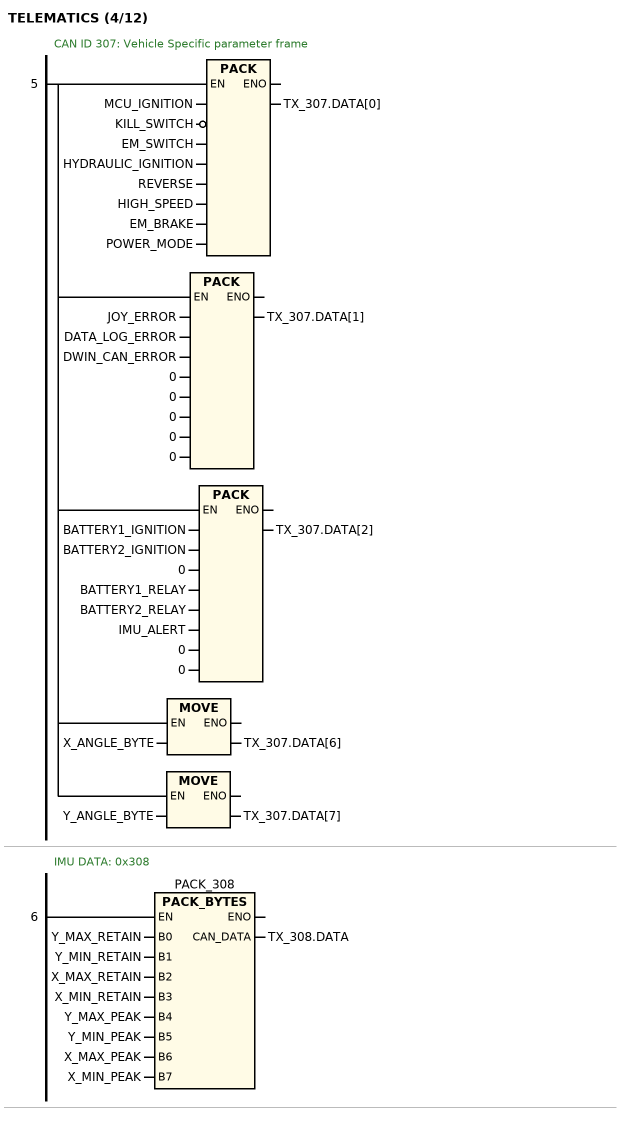
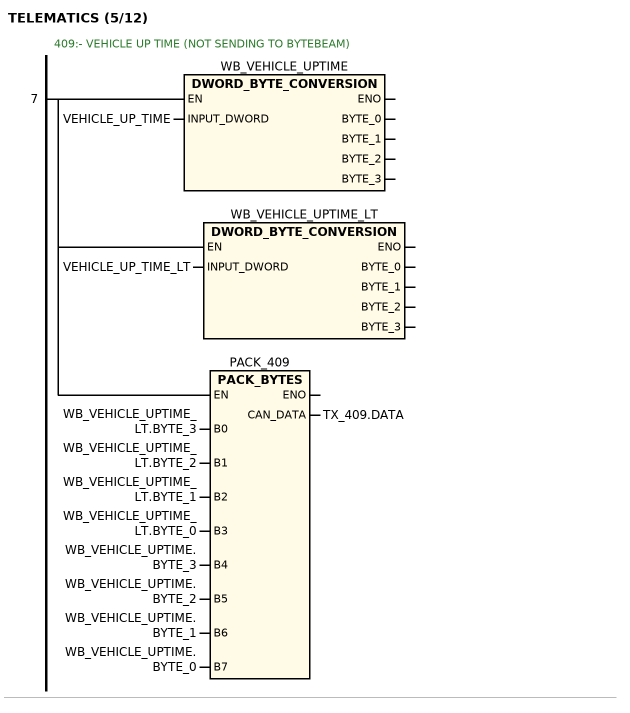
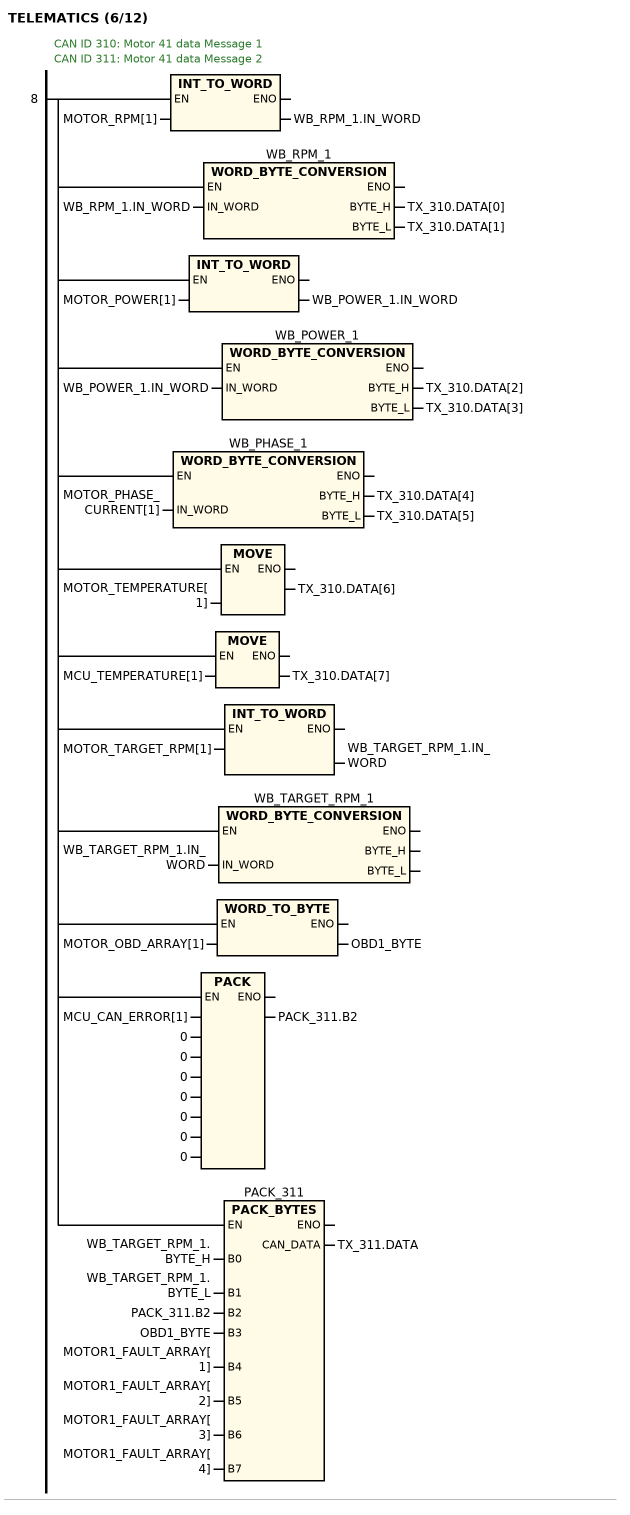
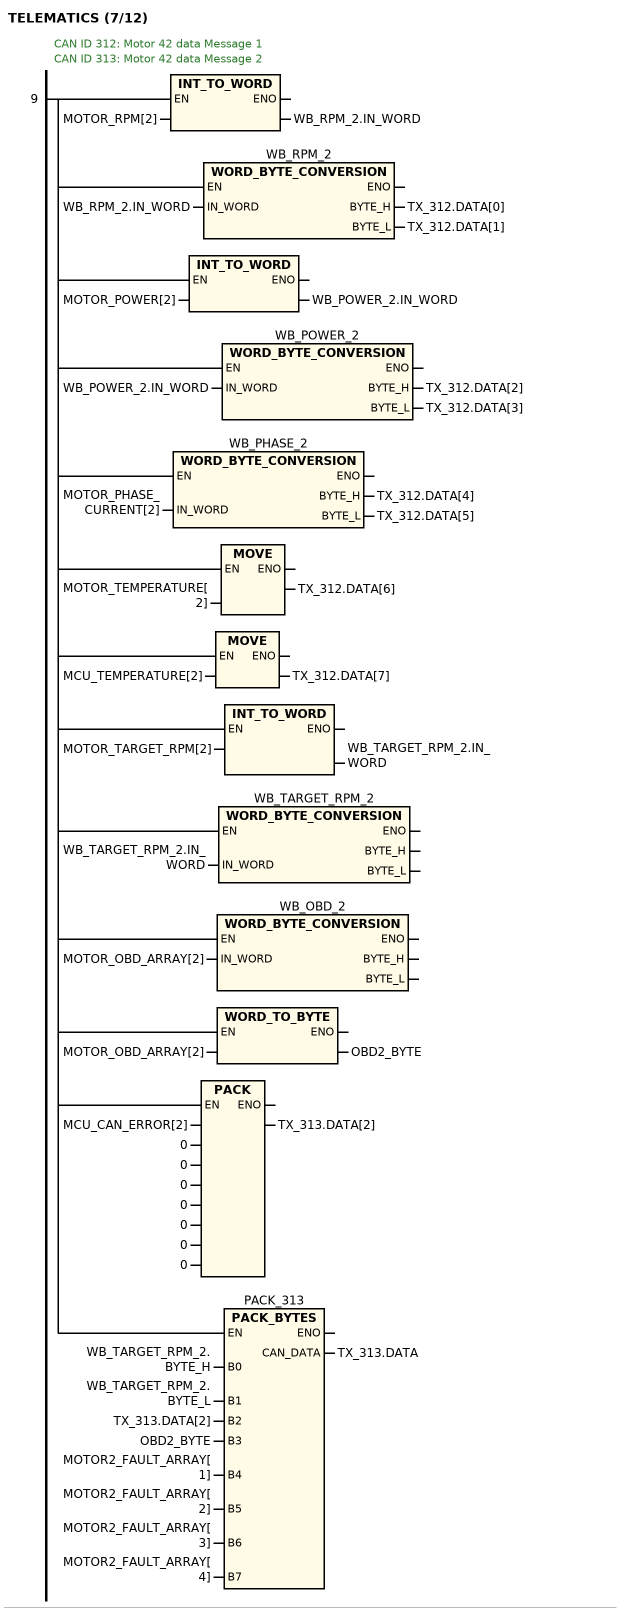
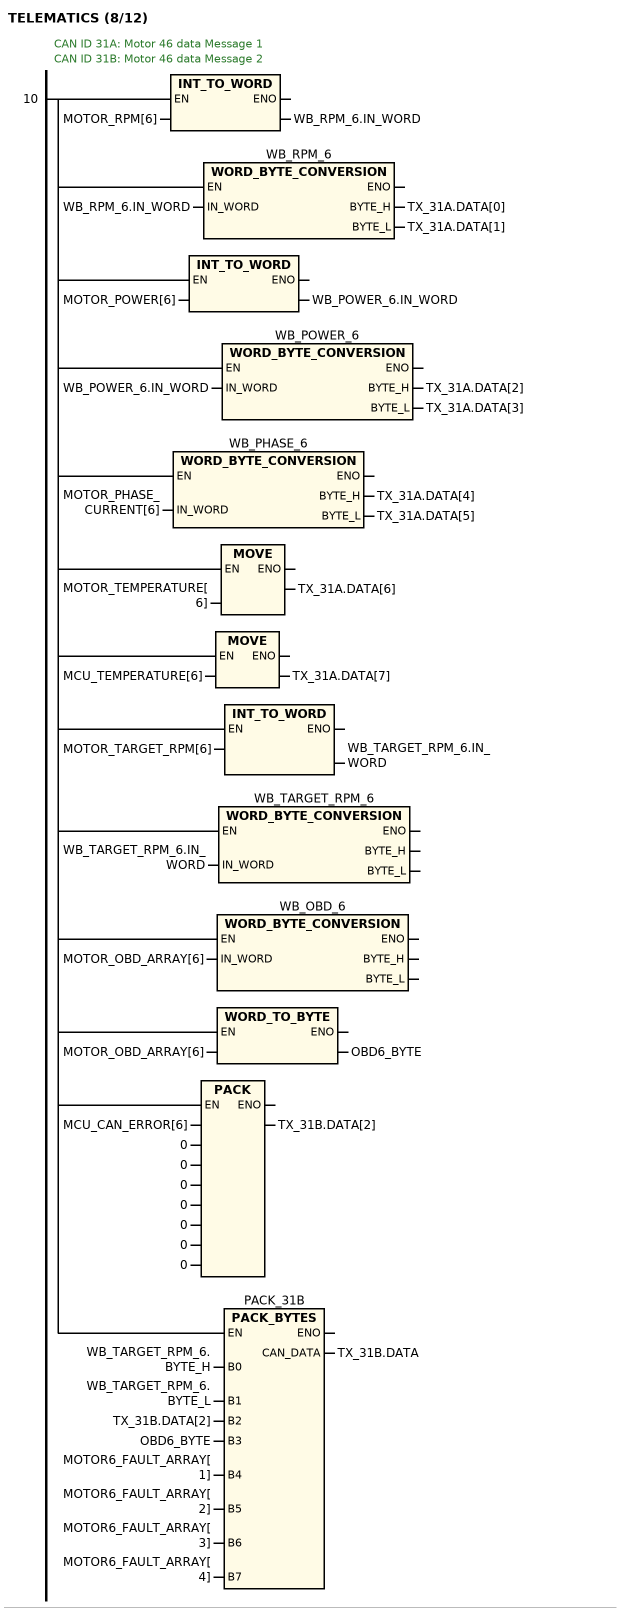
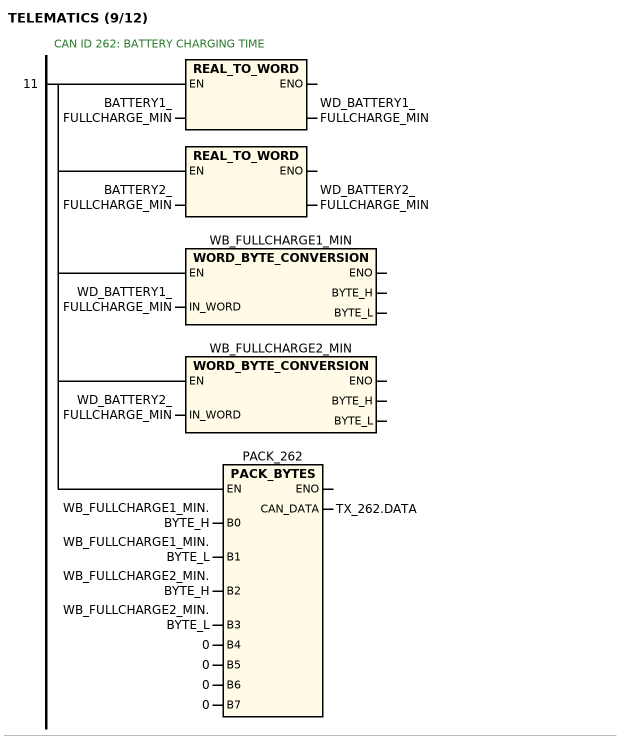
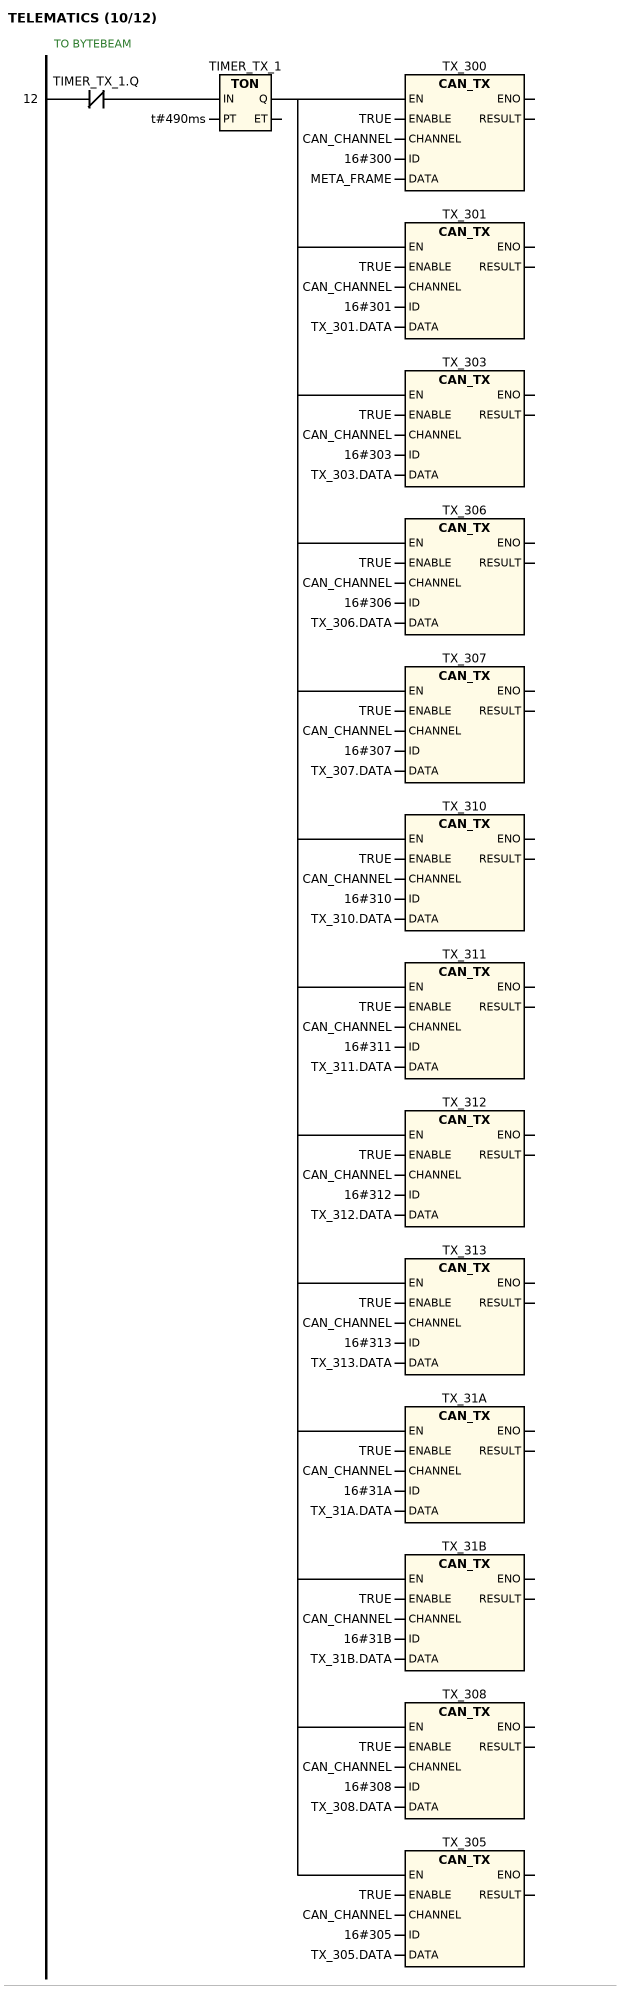
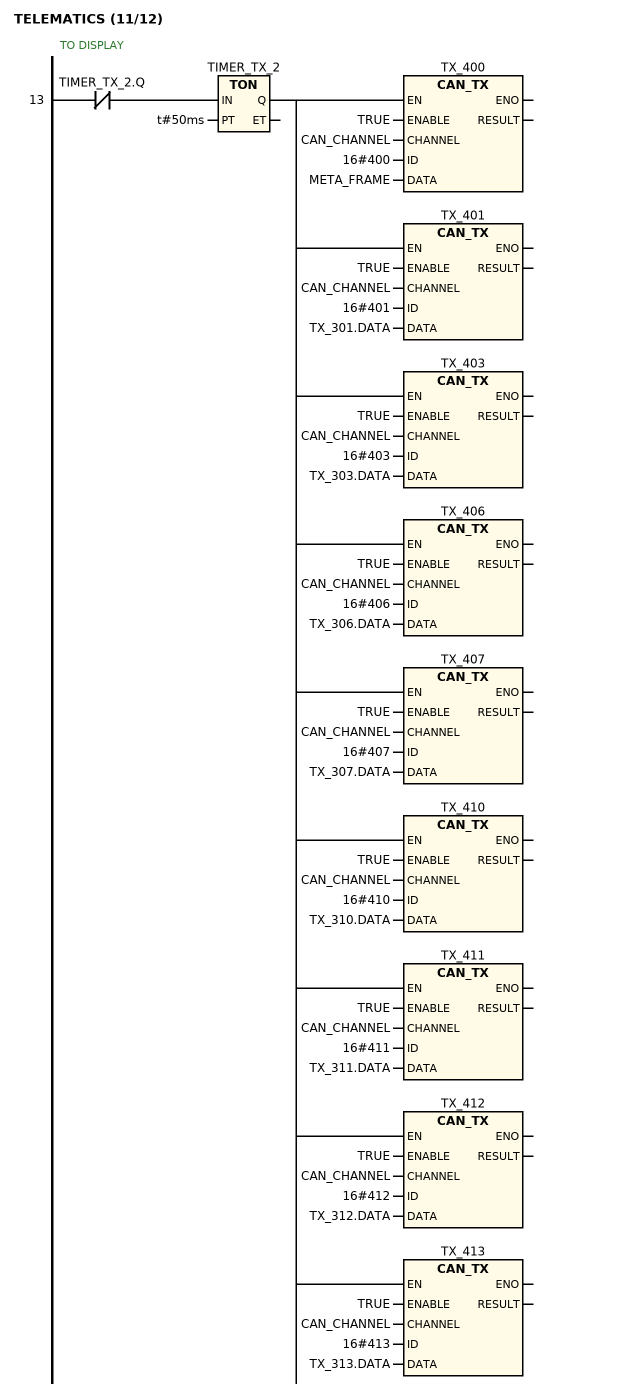
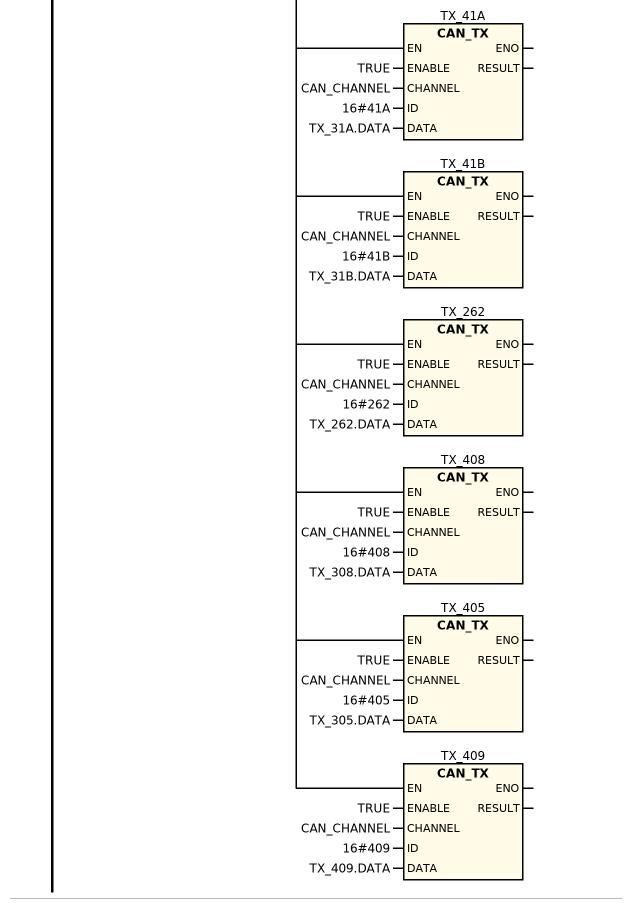
